// Mitsubishi GX Works2 project: Ex   PLC: Q03UDV

PROGRAM MAIN
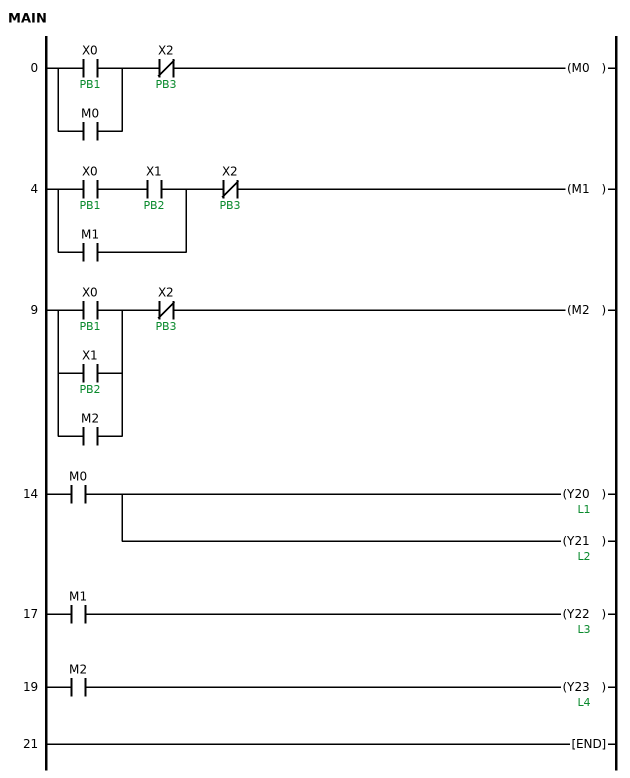
0     LD      X0  ; PB1
      OR      M0
      ANI     X2  ; PB3
      OUT     M0
4     LD      X0  ; PB1
      AND     X1  ; PB2
      OR      M1
      ANI     X2  ; PB3
      OUT     M1
9     LD      X0  ; PB1
      OR      X1  ; PB2
      OR      M2
      ANI     X2  ; PB3
      OUT     M2
14    LD      M0
      OUT     Y20  ; L1
      OUT     Y21  ; L2
17    LD      M1
      OUT     Y22  ; L3
19    LD      M2
      OUT     Y23  ; L4
21    END
END_PROGRAM
